Fanuc KAREL source: kd00005.KL

-- PROVISIONAL review KL for V770-1; original PC SHA256 947eab80aa770f9b135f67dd0a20240b2546b63a06b3340c86ba9aaf52043412
-- Incomplete behavior may be omitted. Consult companion uncertainty JSON. Do not deploy.
PROGRAM KD00005
%NOLOCKGROUP
VAR
  I : INTEGER
  J : INTEGER
  B : BOOLEAN
  R : REAL
  S : STRING[80]
BEGIN
  -- UNRESOLVED_PC offsets 5-12; opcodes 9D,23
  -- UNRESOLVED_PC offsets 17-21; opcodes 7F
END KD00005
